(*
Nazwa:			S_Error
Opis:			Struktura bledu
Wersja:			v0.2
Data:			2018-10-10
Autor:			TW
Urzadzenia:		
Konfiguracja:	
Info:
- dodano string2
*)
TYPE S_Error :
STRUCT
	bError				: BOOL; 
	udiStationID		: UDINT;
	sStationName		: STRING;
	nErrorCode			: UDINT;
	sErrorString		: STRING(200);
	sErrorString2		: STRING(200);
	bReset:BOOL;
END_STRUCT
END_TYPE

(* stored: Version 1.1.0.1, ProductVersion 3.1.4026.13, FileIdentifier 9860c66d2c96fbdee70930f048a4480c1054e1f6, FileSignature 389b337dadb7f3ae58f165d017f5f4af953ddc7e5c2353bc63ebce09f759fc097f023e1f3fe545cd2c71dd39f73af55ac984e934fd0db11bc996ba159e1d0088d111f3ed71081c1d558ee710bf3dde480256f42d740fe17e36399bc59a720ff629b2b09c8c162cf04ede14c814cf849af7d908ef8dfbf758000808a0af44b88474dae343d770666df83e5317479ef01de92ce0444d11a16816475156c3b3324d62efa7666dacd28c64b316673997b481c60e8987a6c8def0ca9151d68b8ebe583f3029fb124341f906283fdd53b54bba24ba34ce5249b410c674cfaf5b70fe484aae168572906e9a9e195262f700e213b7751c6c90fd43b80a60bb82916eb03d
   DUT S_Error: Id {a2465f84-6bc3-478d-a5d4-5472f1bf6aea} *)
